{attribute 'qualified_only'}
{attribute 'strict'}
TYPE KleurmachineToestand :
(
	startup := 0,
	home,
	info,
	scan,
	wachtOpBlik,
	kleurToevoegen,
	klaarMetToevoegen
);
END_TYPE

(* stored: Version 1.1.0.1, ProductVersion 3.1.4024.15
   DUT KleurmachineToestand: Id {5a1a2972-58b5-4eb7-8789-febbb6344c88} *)
